Universal Robots PolyScope program: CircularPath_2.urp

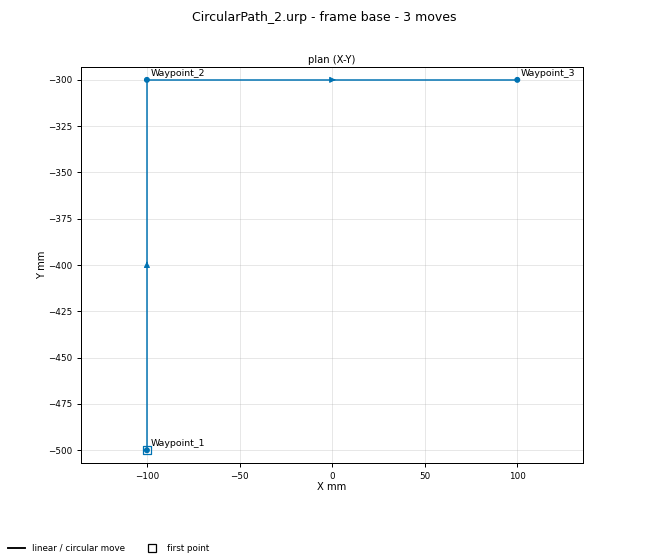
[picture p0: tool path of CircularPath_2.urp in frame base, 3 of 3 moves have a stored position in this frame; points joined in program order, loops and branches not executed]
ProgramRoot directory=/home/ur/ursim-1.5/programs/templates/CircularPathUsingMoveP; kinematics=(a=[0, -0.425, -0.39243, 0, 0, 0], d=[0.0892, 0, 0, 0.109, 0.093, 0.082], alpha=[1.5708, 0, 0, 1.5708, -1.5708, 0], deltaTheta=[0, 0, 0, 0, 0, 0], status=notInitialized); name=CircularPath_2; programVersion=(project__name=PolyScope, major__version=1, minor__version=5, svn__revision=7526, build__date=Dec 21 2011, 13:03:24); robotEnvironmentFileName=default
  MainProgram cartesianAcceleration=1.2; cartesianSpeed=0.25; jointAcceleration=1.3962634015954636; jointSpeed=1.0471975511965976; moveAsFastAsPossible=true; sharedProcessMoveBlendRadius=0.025; featureReference=(installationNameReference=Base); motionType=JOINT_SPACE
    Move cartesianAcceleration=1.2; cartesianSpeed=0.25; jointAcceleration=1.3962634015954636; jointSpeed=1.0471975511965976; moveAsFastAsPossible=true; sharedProcessMoveBlendRadius=0.025; featureReference=(installationNameReference=Base); motionType=PROCESS_MOVE
      Waypoint blendRadius=0.0; cartesianAcceleration=1.2; cartesianSpeed=0.25; jointAcceleration=1.3962634015954636; jointSpeed=1.0471975511965976; nextMotionTime=2.0; useSharedBlendParameter=true; useSharedParameters=true; position=TCP in base x=-100 y=-500 z=200 mm, rx=0 ry=3.14 rz=0.0006 rad; joints [-88.982, -101.255, -113.55, -55.216, 90.094, 1.018] deg; positionType=FIXED_POSITION; waypointPoseInFeatureCoordinates=(pos=(x=-0.09999999999998957, y=-0.5000000000000082, z=0.1999998668199792), rot=(x=-5.308256505009962E-7, y=3.139954578393098, z=6.183385988155127E-4)); name=Waypoint_1
      Waypoint blendRadius=0.05; cartesianAcceleration=1.2; cartesianSpeed=0.25; jointAcceleration=1.3962634015954636; jointSpeed=1.0471975511965976; nextMotionTime=2.0; useSharedParameters=true; position=TCP in base x=-100 y=-300 z=199.999 mm, rx=0 ry=3.14 rz=0.0006 rad; joints [-88.298, -72.82, -140.089, -57.108, 90.094, 1.702] deg; positionType=FIXED_POSITION; waypointPoseInFeatureCoordinates=(pos=(x=-0.10000001312432649, y=-0.3000000004985588, z=0.19999890172054519), rot=(x=-5.831356108308684E-7, y=3.1399538545063836, z=5.547303067392085E-4)); name=Waypoint_2
      Waypoint blendRadius=0.05; cartesianAcceleration=1.2; cartesianSpeed=0.25; jointAcceleration=1.3962634015954636; jointSpeed=1.0471975511965976; nextMotionTime=2.0; stoppoint=true; useSharedBlendParameter=true; useSharedParameters=true; position=TCP in base x=100 y=-300 z=200 mm, rx=0 ry=3.14 rz=0.0006 rad; joints [-51.426, -72.815, -140.108, -57.036, 90.087, 38.574] deg; positionType=FIXED_POSITION; waypointPoseInFeatureCoordinates=(pos=(x=0.09999999999999121, y=-0.2999999999999814, z=0.19999986682001572), rot=(x=-5.308255965683186E-7, y=3.1399545783933682, z=6.183385986190898E-4)); name=Waypoint_3
